PROGRAM MAIN
VAR
END_VAR


RIFD();

END_PROGRAM

(* stored: Version 1.1.0.1
   POU MAIN: Id {351664dc-9997-451d-86c7-99a132d814a0}, SpecialFunc None *)
